// TIA Portal project "Profinet_SR1000_S71200" (V15.1)
// Framework de integracao entre SR1000 e S7-1200 da Siemens, Tia Portal V15.1

(* hardware
DEVICE "SR-1000"  GSD.Device.PN
   slot 0: "Rack"  Rack  V1.0
   slot 0: "sr-1000"  SR-1000X  SR-1000X  1.0
      slot 0: "SR-1000X"  SR-1000X  1.0
      slot 1: "Interface"  Interface
         slot 1: "Port 1"  Port 1
   slot 1: "Handshake and General Error Status Bits_1"  Handshake and General Error Status Bits
      slot 0: "Handshake and General Error Status Bits"  Handshake and General Error Status Bits
   slot 2: "BUSY Status Bits_1"  BUSY Status Bits
      slot 0: "BUSY Status Bits"  BUSY Status Bits
   slot 3: "Completion Status Bits_1"  Completion Status Bits
      slot 0: "Completion Status Bits"  Completion Status Bits
   slot 4: "Error Status Bits_1"  Error Status Bits
      slot 0: "Error Status Bits"  Error Status Bits
   slot 5: "Terminal Status Bits_1"  Terminal Status Bits
      slot 0: "Terminal Status Bits"  Terminal Status Bits
   slot 6: "Unstable Read Status Bits_1"  Unstable Read Status Bits
      slot 0: "Unstable Read Status Bits"  Unstable Read Status Bits
   slot 7: "Matching Level and Total Evaluation Grade Status_1"  Matching Level and Total Evaluation Grade Status
      slot 0: "Matching Level and Total Evaluation Grade Status"  Matching Level and Total Evaluation Grade Status
   slot 8: "Operation Result Status_1"  Operation Result Status
      slot 0: "Operation Result Status"  Operation Result Status
   slot 9: "Read Data 128Byte_1"  Read Data 128Byte
      slot 0: "Read Data 128Byte"  Read Data 128Byte
   slot 10: "Latch and Error Clear Control Bits_1"  Latch and Error Clear Control Bits
      slot 0: "Latch and Error Clear Control Bits"  Latch and Error Clear Control Bits
   slot 11: "Operation instruction Control Bits_1"  Operation instruction Control Bits
      slot 0: "Operation instruction Control Bits"  Operation instruction Control Bits
   slot 12: "Completion Clear Control Bits_1"  Completion Clear Control Bits
      slot 0: "Completion Clear Control Bits"  Completion Clear Control Bits
   slot 13: "Parameter Bank Number_1"  Parameter Bank Number
      slot 0: "Parameter Bank Number"  Parameter Bank Number
   slot 14: "User Data 128Byte_1"  User Data 128Byte
      slot 0: "User Data 128Byte"  User Data 128Byte
DEVICE "PLC 1"  S7-1200 Station
   slot 0: "Rack_0"  S7-1200 Rack  Rack  V1.0
   slot 1: "PLC_1"  CPU 1215C AC/DC/Rly  6ES7 215-1BG40-0XB0  V4.2
*)

// ===== PLC "PLC_1"  CPU 1215C AC/DC/Rly =====

VAR_GLOBAL   // PLC tag table "Default tag table"
   "START TRIGGER" AT %M1.0 : Bool;   // MEMORY TESTE
END_VAR

VAR_GLOBAL   // PLC tag table "SR1000 Tags"
   "Error" AT %I2.0 : Bool;   // Handshake and General Error Status Bits
   "ResultDataAvailable" AT %I2.1 : Bool;   // Handshake and General Error Status Bits
   "ResultDataStrobe" AT %I2.2 : Bool;   // Handshake and General Error Status Bits
   "BufferOverflowError" AT %I2.6 : Bool;   // Handshake and General Error Status Bits
   "General Error" AT %I2.7 : Bool;   // Handshake and General Error Status Bits
   "BUSY" AT %I3.0 : Bool;   // BUSY Status Bits
   "TRG BUSY" AT %I3.1 : Bool;   // BUSY Status Bits
   "LOCK BUSY" AT %I3.2 : Bool;   // BUSY Status Bits
   "MODE BUSY" AT %I3.3 : Bool;   // BUSY Status Bits
   "ERR BUSY" AT %I3.4 : Bool;   // BUSY Status Bits
   "Read Complete" AT %I4.0 : Bool;   // Completion Status Bits
   "Preset Complete" AT %I4.1 : Bool;   // Completion Status Bits
   "RegisterPreset Complete" AT %I4.2 : Bool;   // Completion Status Bits
   "Tune Complete" AT %I4.3 : Bool;   // Completion Status Bits
   "BLOAD Complete" AT %I4.4 : Bool;   // Completion Status Bits
   "EXTRequest Complete" AT %I4.7 : Bool;   // Completion Status Bits
   "Read Failure" AT %I5.0 : Bool;   // Error Status Bits
   "Preset Failure" AT %I5.1 : Bool;   // Error Status Bits
   "RegistPresetFailure" AT %I5.2 : Bool;   // Error Status Bits
   "TuneFailure" AT %I5.3 : Bool;   // Error Status Bits
   "BLOAD Failure" AT %I5.4 : Bool;   // Error Status Bits
   "EXTReqFailure" AT %I5.7 : Bool;   // Error Status Bits
   "IN1" AT %I6.0 : Bool;   // Terminal Status Bits
   "IN2" AT %I6.1 : Bool;   // Terminal Status Bits
   "OUT1" AT %I6.4 : Bool;   // Terminal Status Bits
   "OUT2" AT %I6.5 : Bool;   // Terminal Status Bits
   "OUT3" AT %I6.6 : Bool;   // Terminal Status Bits
   "Unstable" AT %I7.0 : Bool;   // Unstable Read Status Bits
   "MatchingLevelUnstable" AT %I7.1 : Bool;   // Unstable Read Status Bits
   "ISO/IEC15415Unstable" AT %I7.2 : Bool;   // Unstable Read Status Bits
   "AIMDPMUnstable" AT %I7.3 : Bool;   // Unstable Read Status Bits
   "SAEAS9132Unstable" AT %I7.4 : Bool;   // Unstable Read Status Bits
   "MatchingLevel" AT %IW68 : UInt;   // Matching Level and Total Evaluation Grade Status
   "ISO/IEC15415Grade" AT %IW70 : UInt;   // Matching Level and Total Evaluation Grade Status
   "AIMDPMGrade" AT %IW72 : UInt;   // Matching Level and Total Evaluation Grade Status
   "ReadResultCode" AT %IW76 : UInt;   // Operation Result Status
   "PresetResultCode" AT %IW78 : UInt;   // Operation Result Status
   "RegisterPresetDataResultCode" AT %IW80 : UInt;   // Operation Result Status
   "TuneResultCode" AT %IW82 : UInt;   // Operation Result Status
   "BLOAD ResultCode" AT %IW84 : UInt;   // Operation Result Status
   "EXTReqResultCode" AT %IW86 : UInt;   // Operation Result Status
   "GeneralErrorCode" AT %IW88 : UInt;   // Operation Result Status
   "SlaveID" AT %IW96 : UInt;   // Read Data
   "ResultDataReadyCount" AT %IW98 : UInt;   // Read Data
   "ResultDataUpdateCount" AT %IW100 : UInt;   // Read Data
   "ResultDataSize" AT %IW102 : UInt;   // Read Data
   "ResultData0" AT %IB104 : Char;   // Read Data
   "ResultData1" AT %IB105 : Char;   // Read Data
   "ResultData2" AT %IB106 : Char;   // Read Data
   "ResultData3" AT %IB107 : Char;   // Read Data
   "ResultData4" AT %IB108 : Char;   // Read Data
   "ResultData5" AT %IB109 : Char;   // Read Data
   "ResultData6" AT %IB110 : Char;   // Read Data
   "ResultData7" AT %IB111 : Char;   // Read Data
   "ResultData8" AT %IB112 : Char;   // Read Data
   "ResultData9" AT %IB113 : Char;   // Read Data
   "ResultData10" AT %IB114 : Char;   // Read Data
   "ResultData11" AT %IB115 : Char;   // Read Data
   "ResultData12" AT %IB116 : Char;   // Read Data
   "ResultData13" AT %IB117 : Char;   // Read Data
   "ResultData14" AT %IB118 : Char;   // Read Data
   "ResultData15" AT %IB119 : Char;   // Read Data
   "Result Data Latch" AT %Q2.1 : Bool;   // Latch and Error Clear Control Bits
   "ErrorClear" AT %Q2.7 : Bool;   // Latch and Error Clear Control Bits
   "Read Request" AT %Q3.0 : Bool;   // Operation instruction Control Bits
   "Preset Request" AT %Q3.1 : Bool;   // Operation instruction Control Bits
   "RegisterPresetDataReq" AT %Q3.2 : Bool;   // Operation instruction Control Bits
   "TuneRequest" AT %Q3.3 : Bool;   // Operation instruction Control Bits
   "BLOAD Request" AT %Q3.4 : Bool;   // Operation instruction Control Bits
   "Read CompleteClear" AT %Q4.0 : Bool;   // Completion Clear Control Bits
   "Preset CompleteClear" AT %Q4.1 : Bool;   // Completion Clear Control Bits
   "RegisterPresetDataCmpltClr" AT %Q4.2 : Bool;   // Completion Clear Control Bits
   "TuneCmpltClr" AT %Q4.3 : Bool;   // Completion Clear Control Bits
   "BLOAD CmpltClr" AT %Q4.4 : Bool;   // Completion Clear Control Bits
   "EXTReqCmpltClr" AT %Q4.7 : Bool;   // Completion Clear Control Bits
   "BankNo" AT %QW68 : UInt;   // Parameter Bank Number
   "UserDataSize" AT %QW70 : UInt;   // User Data
   "UserData0" AT %QB72 : Char;   // User Data
   "UserData1" AT %QB73 : Char;   // User Data
   "UserData2" AT %QB74 : Char;   // User Data
   "UserData3" AT %QB75 : Char;   // User Data
   "UserData4" AT %QB76 : Char;   // User Data
   "UserData5" AT %QB77 : Char;   // User Data
   "UserData6" AT %QB78 : Char;   // User Data
   "UserData7" AT %QB79 : Char;   // User Data
   "UserData8" AT %QB80 : Char;   // User Data
   "UserData9" AT %QB81 : Char;   // User Data
   "UserData10" AT %QB82 : Char;   // User Data
   "UserData11" AT %QB83 : Char;   // User Data
   "UserData12" AT %QB84 : Char;   // User Data
   "UserData13" AT %QB85 : Char;   // User Data
   "UserData14" AT %QB86 : Char;   // User Data
   "UserData15" AT %QB87 : Char;   // User Data
END_VAR

FUNCTION "SR-1000" : Void   // FC1, LAD
TITLE = SR-1000
{ S7_Optimized_Access := 'TRUE' }
VERSION : 0.1
BEGIN

REGION Network 1: REQUESICAO PARA DISPARO
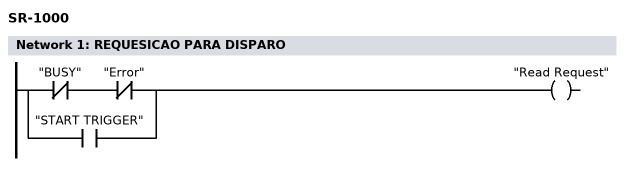
   RUNG wire#powerrail
      I_Contact( "BUSY" )
      I_Contact( "Error" )
      wire#w1
      Coil( "Read Request" )
   END_RUNG
   RUNG wire#powerrail
      Contact( "START TRIGGER" )
   END_RUNG wire#w1
   // the same network as SCL:
   "Read Request" := (NOT "BUSY" AND NOT "Error") OR "START TRIGGER";
END_REGION
END_FUNCTION

ORGANIZATION_BLOCK "Main"   // OB1, LAD, ProgramCycle
TITLE = "Main Program Sweep (Cycle)"
{ S7_Optimized_Access := 'TRUE' }
VERSION : 0.1
   VAR_INPUT
      Initial_Call : Bool;   // Initial call of this OB
      Remanence : Bool;   // =True, if remanent data are available
   END_VAR
BEGIN

REGION Network 1: CHAMADA FC1 - SR-1000
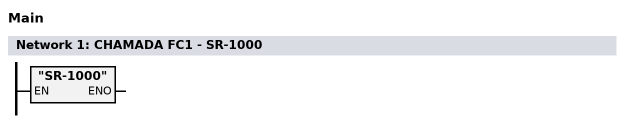
   RUNG wire#powerrail
      "SR-1000"()
   END_RUNG
   // the same network as SCL:
   "SR-1000"();
END_REGION
END_ORGANIZATION_BLOCK